TYPE "SpeedMachine_Par"
VERSION : 0.1
// Block: SpeedMachine_Par
   STRUCT
      Man : Struct
         VelBwd : LReal;
         VelFwdHigh : LReal;
         VelFwdLow : LReal;
         Acc : LReal;
         Dec : LReal;
         DelayChangeVel : Time;
      END_STRUCT;
   END_STRUCT;

END_TYPE
